Universal Robots PolyScope program: ejemplo_pose_add.urp

Program ejemplo_pose_add (installation=default directory=/home/ur/ursim-current/programs createdIn=3.6.1.30595 lastSavedIn=3.14.3.1031232 robotSerialNumber=2018339999)
Calibrated DH parameters: a=[0, -0.24365, -0.21325, 0, 0, 0]; d=[0.1519, 0, 0, 0.11235, 0.08535, 0.0819]; alpha=[1.570796, 0, 0, 1.570796, -1.570796, 0]; deltaTheta=[0, 0, 0, 0, 0, 0]
Robot Program (runOnlyOnce=true)
  MoveJ speed 60 deg/s, acceleration 80 deg/s^2 (useActiveTCP=true)
    SuppressedNode
      Waypoint Punto_de_paso_1: TCP in base x=-299.976 y=150.002 z=0.009 mm, rx=3.14 ry=0 rz=0.0001 rad; joints [-187.092, -95.607, -98.16, -76.247, 90.089, 82.907] deg; flange x=-299.985 y=150.411 z=261.719 mm, rx=3.14 ry=0 rz=0.0001 rad
    P_ini := get_actual_tcp_pose()
    SuppressedNode
      punto_ref := p[-0.3,0.15,0,3.14,0,0]
    Waypoint Waypoint (Variable): variable=P_ini
    Wait Sleep waitTime=1
    x := 100
    y := 120
    z1 := -100
    rx := 0
    ry := 0
    rz := 0
    desplazamiento := p[x/1000,y/1000,z1/1000,rx,ry,rz]
    pos_coger := pose_add(P_ini,desplazamiento)
  MoveL speed 250 mm/s, acceleration 1200 mm/s^2 (useActiveTCP=true) feature=Base
    Waypoint Waypoint (Variable): variable=pos_coger
    Wait Sleep waitTime=2
  Halt
